///////////
// Structure For Battery Racks. Main Operating Data to be saved ( ex: OPC ) .  
//////////
TYPE Cell :
STRUCT
	MesU			: REAL ;    		(*( V) Cell voltage *)
	
END_STRUCT
END_TYPE

(* stored: Version 1.1.0.1, ProductVersion 3.1.4024.6
   DUT Cell: Id {b36c54e5-e6de-434b-ab93-bc2ecbe9062c} *)
